FUNCTION_BLOCK "LAnyAxis_MC_CamIn"
{ S7_Optimized_Access := 'TRUE' }
AUTHOR : 'tech.team.motioncontrol@siemens.com'
FAMILY : AnyAxis
VERSION : 1.0
   VAR_INPUT
      Master : DB_ANY;
      Slave : DB_ANY;
      Cam : DB_ANY;
      Execute : Bool;
      MasterOffset : LReal;
      SlaveOffset : LReal;
      MasterScaling : LReal := 1.0;
      SlaveScaling : LReal := 1.0;
      MasterSyncPosition : LReal;
      SyncProfileReference : DInt := 1;
      MasterStartDistance : LReal;
      Velocity : LReal := -1.0;
      Acceleration : LReal := -1.0;
      Deceleration : LReal := -1.0;
      Jerk : LReal := -1.0;
      ApplicationMode : DInt;
      SyncDirection : DInt := 3;
   END_VAR

   VAR_OUTPUT
      StartSync { ExternalWritable := 'False'} : Bool := FALSE;
      InSync { ExternalWritable := 'False'} : Bool := FALSE;
      Busy { ExternalWritable := 'False'} : Bool := FALSE;
      CommandAborted { ExternalWritable := 'False'} : Bool := FALSE;
      Error { ExternalWritable := 'False'} : Bool := FALSE;
      ErrorId { ExternalWritable := 'False'} : Word := 16#0000;
      EndOfProfile { ExternalWritable := 'False'} : Bool;
   END_VAR

   VAR
      instMC {InstructionName := 'MC_CAMIN'; LibVersion := '5.0'; ExternalAccessible := 'False'; ExternalVisible := 'False'; ExternalWritable := 'False'; S7_SetPoint := 'False'} : MC_CAMIN;
      statExecuteOld { ExternalAccessible := 'False'; ExternalVisible := 'False'; ExternalWritable := 'False'} : Bool;
      statAxis { ExternalAccessible := 'False'; ExternalVisible := 'False'; ExternalWritable := 'False'} : DB_ANY;
      statAxisType { ExternalAccessible := 'False'; ExternalVisible := 'False'; ExternalWritable := 'False'} : Int;
      statMaster { ExternalAccessible := 'False'; ExternalVisible := 'False'; ExternalWritable := 'False'} : DB_ANY;
      statMasterType { ExternalAccessible := 'False'; ExternalVisible := 'False'; ExternalWritable := 'False'} : Int;
      statCam { ExternalAccessible := 'False'; ExternalVisible := 'False'; ExternalWritable := 'False'} : DB_ANY;
   END_VAR

   VAR CONSTANT
      ERROR_INVALID_TECHNOLOGY_OBJECT : Word := 16#8002;
      IDLE : Int := 0;
      INVALID_AXIS : Int := -1;
      INVALID_MASTER : Int := -2;
      INVALID_CAM : Int := -3;
      EXTERNAL_ENCODER : Int := 1;
      POSITIONING_AXIS : Int := 3;
      SYNCHRONOUS_AXIS : Int := 4;
      PROXY : Int := 5;
   END_VAR


BEGIN
	REGION HEADER
	  //================================================================================
	  // SIEMENS AG
	  // (c)Copyright 2020 All Rights Reserved
	  //--------------------------------------------------------------------------------
	  // Library: LAnyAxis
	  // Tested with: S7-1515T-2 PN
	  // Engineering: TIA Portal V16
	  // Restrictions: -
	  // Requirements: S7-1500T FW 2.8.1
	  // Functionality: Conversion DB_ANY --> TO_Axis
	  // Support: tech.team.motioncontrol@siemens.com
	  // Note: Parameter comments are only available in language 'English (United States)'
	  //--------------------------------------------------------------------------------
	  // Change log table:
	  // Version  Date        Expert in charge  Changes applied
	  // 01.00.00 10.03.2020  RS                First released version
	  //================================================================================
	END_REGION

	REGION EXECUTE
	  IF #Execute AND NOT #statExecuteOld THEN
	    // Copy parameter
	    #instMC.MasterOffset := #MasterOffset;
	    #instMC.SlaveOffset := #SlaveOffset;
	    #instMC.MasterScaling := #MasterScaling;
	    #instMC.SlaveScaling := #SlaveScaling;
	    #instMC.MasterSyncPosition := #MasterSyncPosition;
	    #instMC.SyncProfileReference := #SyncProfileReference;
	    #instMC.MasterStartDistance := #MasterStartDistance;
	    #instMC.Velocity := #Velocity;
	    #instMC.Acceleration := #Acceleration;
	    #instMC.Deceleration := #Deceleration;
	    #instMC.Jerk := #Jerk;
	    #instMC.ApplicationMode := #ApplicationMode;
	    #instMC.SyncDirection := #SyncDirection;

	    // Check axis type
	    CASE TypeOfDB(#Slave) OF
	      TO_SYNCHRONOUSAXIS:
	        #statAxisType := #SYNCHRONOUS_AXIS;
	        #statAxis := #Slave;

	        // Check master type
	        CASE TypeOfDB(#Master) OF
	          TO_POSITIONINGAXIS:
	            #statMasterType := #POSITIONING_AXIS;
	            #statMaster := #Master;

	          TO_SYNCHRONOUSAXIS:
	            #statMasterType := #SYNCHRONOUS_AXIS;
	            #statMaster := #Master;

	          TO_EXTERNALENCODER:
	            #statMasterType := #EXTERNAL_ENCODER;
	            #statMaster := #Master;

	          TO_LEADINGAXISPROXY:
	            #statMasterType := #PROXY;
	            #statMaster := #Master;
	          ELSE
	            #statMasterType := #INVALID_AXIS;
	            #statMaster := 0;

	            // Invalid master
	            #statAxisType := #INVALID_MASTER;
	        END_CASE;

	      ELSE
	        #statAxisType := #INVALID_AXIS;
	        #statAxis := 0;
	    END_CASE;

	    IF (TypeOfDB(#Cam) = TO_Cam) THEN
	      #statCam := #Cam;
	    ELSE
	      #statCam := 0;
	      #statAxisType := #INVALID_CAM;
	    END_IF;

	  ELSIF NOT #Execute AND (#statAxisType < #IDLE) THEN
	    #statAxisType := #IDLE;

	    // Outputs
	    #StartSync := FALSE;
	    #InSync := FALSE;
	    #Busy := FALSE;
	    #CommandAborted := FALSE;
	    #Error := FALSE;
	    #ErrorId := 16#0000;
	    #EndOfProfile := FALSE;
	  END_IF;

	  // Edge detection
	  #statExecuteOld := #Execute;
	END_REGION

	CASE #statAxisType OF
	  #IDLE:
	    ;

	  #SYNCHRONOUS_AXIS:
	    REGION VALID_AXIS
	      // Inputs
	      #instMC.Execute := #Execute;

	      // Call of MC instruction
	      CASE #statMasterType OF
	        #POSITIONING_AXIS:
	          "LAnyAxis_UnpubCamInMasterPosAxis"(slave := #statAxis,
	                                             master := #statMaster,
	                                             cam := #Cam,
	                                             instMC := #instMC);
	        #SYNCHRONOUS_AXIS:
	          "LAnyAxis_UnpubCamInMasterSyncAxis"(slave := #statAxis,
	                                              master := #statMaster,
	                                              cam := #Cam,
	                                              instMC := #instMC);
	        #EXTERNAL_ENCODER:
	          "LAnyAxis_UnpubCamInMasterExtEncoder"(slave := #statAxis,
	                                                master := #statMaster,
	                                                cam := #Cam,
	                                                instMC := #instMC);
	        #PROXY:
	          "LAnyAxis_UnpubCamInMasterProxy"(slave := #statAxis,
	                                           master := #statMaster,
	                                           cam := #Cam,
	                                           instMC := #instMC);
	      END_CASE;

	      // Outputs
	      #StartSync := #instMC.StartSync;
	      #InSync := #instMC.InSync;
	      #Busy := #instMC.Busy;
	      #CommandAborted := #instMC.CommandAborted;
	      #Error := #instMC.Error;
	      #ErrorId := #instMC.ErrorId;
	      #EndOfProfile := #instMC.EndOfProfile;

	      // Status of MC instruction
	      IF NOT #instMC.Busy
	        AND NOT #instMC.CommandAborted
	        AND NOT #instMC.Error
	        AND NOT #instMC.EndOfProfile
	      THEN
	        // Not active
	        #statAxisType := #IDLE;
	      END_IF;
	    END_REGION
	  ELSE
	    REGION INVALID_TECHNOLOGY_OBJECT
	      // Outputs
	      #StartSync := FALSE;
	      #InSync := FALSE;
	      #Busy := FALSE;
	      #CommandAborted := FALSE;
	      #Error := TRUE;
	      #ErrorId := #ERROR_INVALID_TECHNOLOGY_OBJECT;
	      #EndOfProfile := FALSE;
	    END_REGION
	END_CASE;
END_FUNCTION_BLOCK

